{attribute 'qualified_only'}
VAR_GLOBAL
	
	//define messages for machine base
	gMsgMc	:typeStationMessage;
	
	//define message for each station
	gMsgS1	:typeStationMessage;
	gMsgS2	:typeStationMessage;
	gMsgS3	:typeStationMessage;
	gMsgS4	:typeStationMessage;
	gMsgS5	:typeStationMessage;
	gMsgS6	:typeStationMessage;
	
	//global memory for retaining status of station
	gMsgMcStat	:typeStationStatus;
	gMsgS1Stat	:typeStationStatus;
	gMsgS2Stat	:typeStationStatus;
	gMsgS3Stat	:typeStationStatus;
	gMsgS4Stat	:typeStationStatus;
	gMsgS5Stat	:typeStationStatus;
	gMsgS6Stat	:typeStationStatus;
	
	//list view of messages in array form
	gListMsgMc	:typeMessageRowsArry;
	gListMsgS1	:typeMessageRowsArry;
	gListMsgS2	:typeMessageRowsArry;
	gListMsgS3	:typeMessageRowsArry;
	gListMsgS4	:typeMessageRowsArry;
	gListMsgS5	:typeMessageRowsArry;
	gListMsgS6	:typeMessageRowsArry;

	gAnyFaultMessage: BOOL; //TRUE if there are any fault messages (any)
	gAnyWarnings: BOOL; //TRUE if there are any warnings (the yellow ones)



	
	
END_VAR


VAR_GLOBAL CONSTANT
	
		AllocMsgPerRow:UINT := 10; //number of messages assigned per row
		gNumMessagesPerType:INT := 1000; //number of messages in each type of message
END_VAR

(* stored: Version 1.1.0.1, ProductVersion 3.1.4024.12
   GVL GlobalMessages: Id {0ab881e6-f244-4b39-9d1f-44ab679d9a69} *)
